INTERFACE ITF_EM_Transport_Checkweigher_BottomSeal

END_INTERFACE

(* stored: Version 1.1.0.1, ProductVersion 3.1.4024.12
   Itf ITF_EM_Transport_Checkweigher_BottomSeal: Id {443d4f44-1a2a-4eec-bbcc-af005769f18b} *)
